// TIA Portal V15.1 export
// export: Created 2024-05-17T05:39:00.3704573Z, ExportSetting WithDefaults, DisplayName Totally Integrated Automation Portal, DisplayVersion V15.1 Update 5, DisplayName TIA Portal Openness, DisplayVersion V15.1 Update 5, DisplayName SINAMICS Startdrive Advanced, DisplayVersion V15.1, DisplayName G130, G150, S120, S150, SINAMICS MV, S210, DisplayVersion V15.1, DisplayName G110M, G120, G120C, G120D, G120P, DisplayVersion V15.1, DisplayName STEP 7 Professional, DisplayVersion V15.1 Update 5, DisplayName STEP 7 Safety, DisplayVersion V15.1, DisplayName WinCC Professional, DisplayVersion V15.1 Update 5, DisplayName SIMATIC Visualization Architect, DisplayVersion V15.1
FUNCTION "209000NCP01AE" : Void   // FC253, FBD
TITLE = 209000NCP01AE
{ S7_Optimized_Access := 'FALSE' }
AUTHOR : VCC
NAME : LocFnc
VERSION : 0.1
// stored: AutoNumber false, IsIECCheckEnabled false, SetENOAutomatically False, UDAEnableTagReadback false
   VAR_OUTPUT
      O_AlarmA : Bool;   // Alarm A
      O_AlarmB : Bool;   // Alarm B
      O_AlarmC : Bool;   // Alarm C
      O_AlarmD : Bool;   // Alarm D
      O_AlarmABCondition : Bool;   // Alarms resetable
      H_IAnim : Word;   // For animation of icon
   END_VAR
BEGIN

REGION Network 1: **** --------------------- AE01 --------------------- ****
END_REGION

REGION Network 2: **** 2.2 Alarms - Alarm generation **** AE01E1QM1 - AE01 EG1 - Overload protection power supply 24VDC
   // AE01 EG1 - Overload protection power supply 24VDC
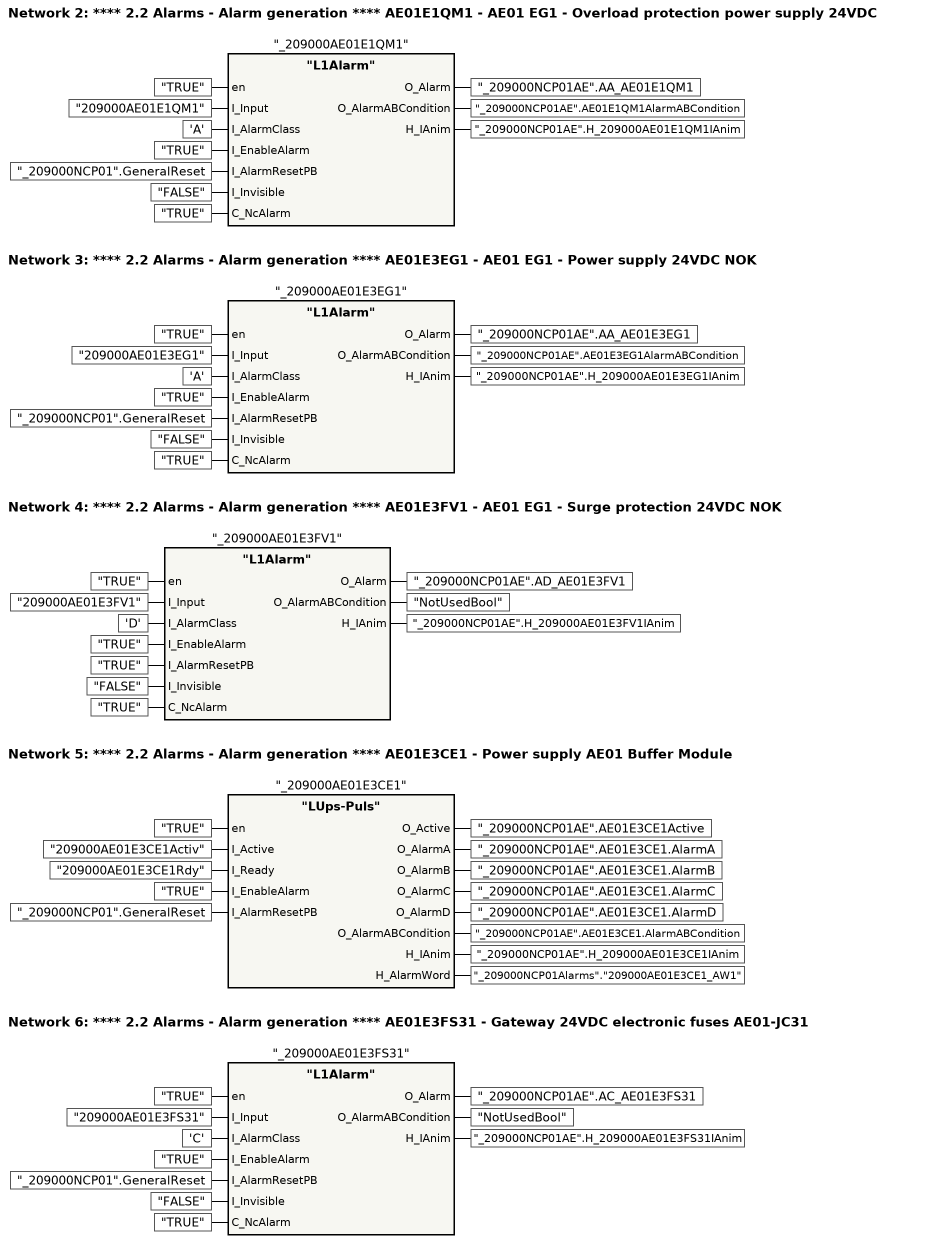
   IF "TRUE" THEN
       "_209000AE01E1QM1"(I_Input := "209000AE01E1QM1",   // "L1Alarm"
                          I_AlarmClass := 'A',
                          I_EnableAlarm := "TRUE",
                          I_AlarmResetPB := "_209000NCP01".GeneralReset,
                          I_Invisible := "FALSE",
                          C_NcAlarm := "TRUE",
                          O_Alarm => "_209000NCP01AE".AA_AE01E1QM1,
                          O_AlarmABCondition => "_209000NCP01AE".AE01E1QM1AlarmABCondition,
                          H_IAnim => "_209000NCP01AE".H_209000AE01E1QM1IAnim);
   END_IF;
END_REGION

REGION Network 3: **** 2.2 Alarms - Alarm generation **** AE01E3EG1 - AE01 EG1 - Power supply 24VDC NOK
   // AE01 EG1 - Power supply 24VDC NOK
   IF "TRUE" THEN
       "_209000AE01E3EG1"(I_Input := "209000AE01E3EG1",   // "L1Alarm"
                          I_AlarmClass := 'A',
                          I_EnableAlarm := "TRUE",
                          I_AlarmResetPB := "_209000NCP01".GeneralReset,
                          I_Invisible := "FALSE",
                          C_NcAlarm := "TRUE",
                          O_Alarm => "_209000NCP01AE".AA_AE01E3EG1,
                          O_AlarmABCondition => "_209000NCP01AE".AE01E3EG1AlarmABCondition,
                          H_IAnim => "_209000NCP01AE".H_209000AE01E3EG1IAnim);
   END_IF;
END_REGION

REGION Network 4: **** 2.2 Alarms - Alarm generation **** AE01E3FV1 - AE01 EG1 - Surge protection 24VDC NOK
   // AE01 EG1 - Surge protection 24VDC NOK
   IF "TRUE" THEN
       "_209000AE01E3FV1"(I_Input := "209000AE01E3FV1",   // "L1Alarm"
                          I_AlarmClass := 'D',
                          I_EnableAlarm := "TRUE",
                          I_AlarmResetPB := "TRUE",
                          I_Invisible := "FALSE",
                          C_NcAlarm := "TRUE",
                          O_Alarm => "_209000NCP01AE".AD_AE01E3FV1,
                          O_AlarmABCondition => "NotUsedBool",
                          H_IAnim => "_209000NCP01AE".H_209000AE01E3FV1IAnim);
   END_IF;
END_REGION

REGION Network 5: **** 2.2 Alarms - Alarm generation **** AE01E3CE1 - Power supply AE01 Buffer Module
   // Power supply  AE01 Buffer Module
   IF "TRUE" THEN
       "_209000AE01E3CE1"(I_Active := "209000AE01E3CE1Activ",   // "LUps-Puls"
                          I_Ready := "209000AE01E3CE1Rdy",
                          I_EnableAlarm := "TRUE",
                          I_AlarmResetPB := "_209000NCP01".GeneralReset,
                          O_Active => "_209000NCP01AE".AE01E3CE1Active,
                          O_AlarmA => "_209000NCP01AE".AE01E3CE1.AlarmA,
                          O_AlarmB => "_209000NCP01AE".AE01E3CE1.AlarmB,
                          O_AlarmC => "_209000NCP01AE".AE01E3CE1.AlarmC,
                          O_AlarmD => "_209000NCP01AE".AE01E3CE1.AlarmD,
                          O_AlarmABCondition => "_209000NCP01AE".AE01E3CE1.AlarmABCondition,
                          H_IAnim => "_209000NCP01AE".H_209000AE01E3CE1IAnim,
                          H_AlarmWord => "_209000NCP01Alarms"."209000AE01E3CE1_AW1");
   END_IF;
END_REGION

REGION Network 6: **** 2.2 Alarms - Alarm generation **** AE01E3FS31 - Gateway 24VDC electronic fuses AE01-JC31
   // Gateway 24VDC electronic fuses AE01-JC31
   IF "TRUE" THEN
       "_209000AE01E3FS31"(I_Input := "209000AE01E3FS31",   // "L1Alarm"
                           I_AlarmClass := 'C',
                           I_EnableAlarm := "TRUE",
                           I_AlarmResetPB := "_209000NCP01".GeneralReset,
                           I_Invisible := "FALSE",
                           C_NcAlarm := "TRUE",
                           O_Alarm => "_209000NCP01AE".AC_AE01E3FS31,
                           O_AlarmABCondition => "NotUsedBool",
                           H_IAnim => "_209000NCP01AE".H_209000AE01E3FS31IAnim);
   END_IF;
END_REGION

REGION Network 7: **** 2.2 Alarms - Alarm generation **** AE01E3FS01 // CH1 - 24VDC Fuse - General - PLC
   // 24VDC Fuse - General - PLC
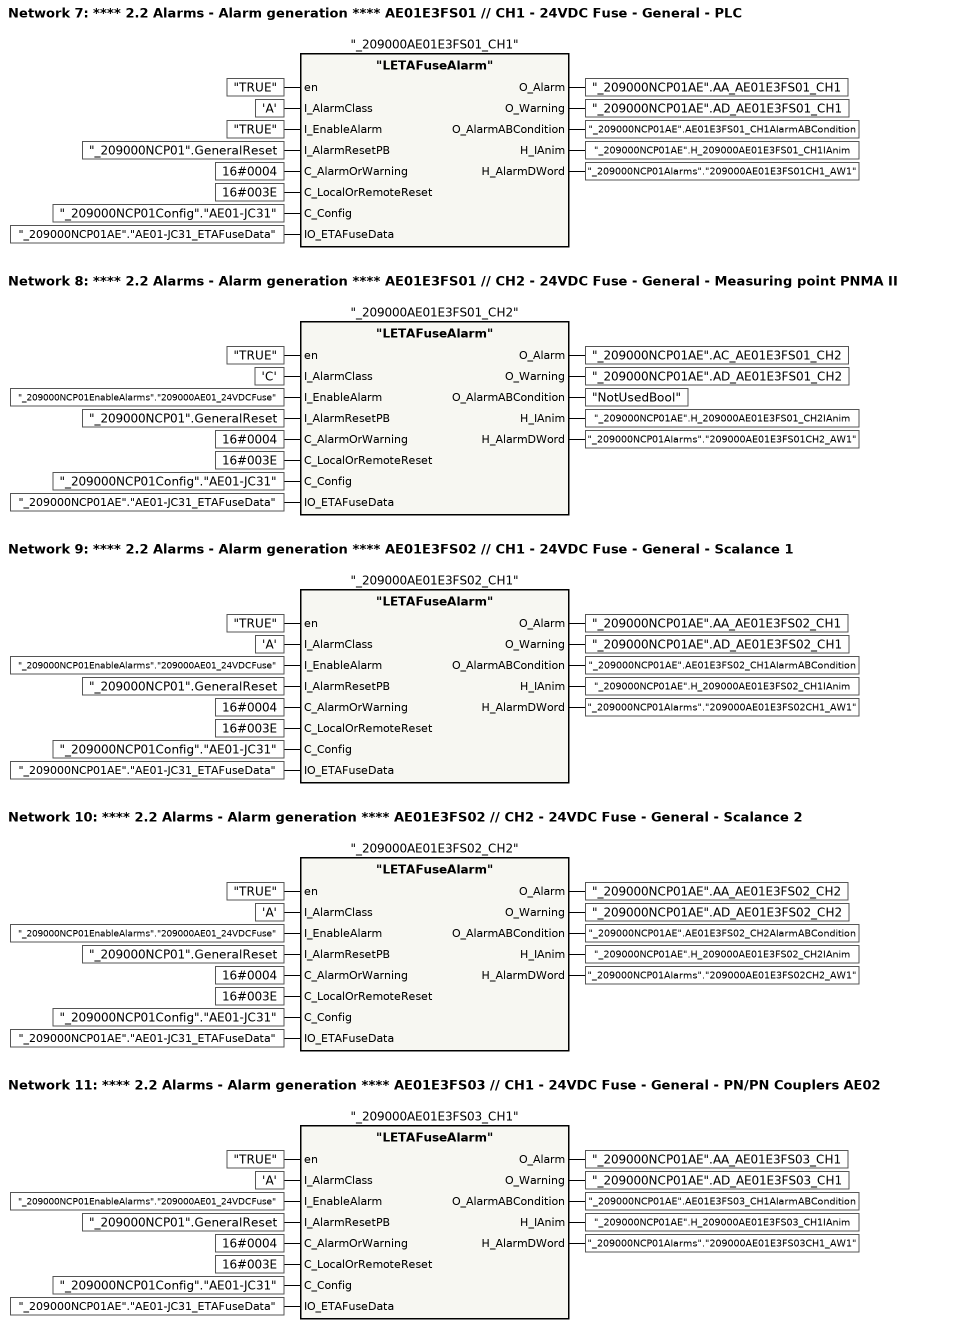
   IF "TRUE" THEN
       "_209000AE01E3FS01_CH1"(I_AlarmClass := 'A',   // "LETAFuseAlarm"
                               I_EnableAlarm := "TRUE",
                               I_AlarmResetPB := "_209000NCP01".GeneralReset,
                               C_AlarmOrWarning := 16#0004,
                               C_LocalOrRemoteReset := 16#003E,
                               C_Config := "_209000NCP01Config"."AE01-JC31",
                               IO_ETAFuseData := "_209000NCP01AE"."AE01-JC31_ETAFuseData",
                               O_Alarm => "_209000NCP01AE".AA_AE01E3FS01_CH1,
                               O_Warning => "_209000NCP01AE".AD_AE01E3FS01_CH1,
                               O_AlarmABCondition => "_209000NCP01AE".AE01E3FS01_CH1AlarmABCondition,
                               H_IAnim => "_209000NCP01AE".H_209000AE01E3FS01_CH1IAnim,
                               H_AlarmDWord => "_209000NCP01Alarms"."209000AE01E3FS01CH1_AW1");
   END_IF;
END_REGION

REGION Network 8: **** 2.2 Alarms - Alarm generation **** AE01E3FS01 // CH2 - 24VDC Fuse - General - Measuring point PNMA II
   // 24VDC Fuse - General - Measuring point PNMA II
   IF "TRUE" THEN
       "_209000AE01E3FS01_CH2"(I_AlarmClass := 'C',   // "LETAFuseAlarm"
                               I_EnableAlarm := "_209000NCP01EnableAlarms"."209000AE01_24VDCFuse",
                               I_AlarmResetPB := "_209000NCP01".GeneralReset,
                               C_AlarmOrWarning := 16#0004,
                               C_LocalOrRemoteReset := 16#003E,
                               C_Config := "_209000NCP01Config"."AE01-JC31",
                               IO_ETAFuseData := "_209000NCP01AE"."AE01-JC31_ETAFuseData",
                               O_Alarm => "_209000NCP01AE".AC_AE01E3FS01_CH2,
                               O_Warning => "_209000NCP01AE".AD_AE01E3FS01_CH2,
                               O_AlarmABCondition => "NotUsedBool",
                               H_IAnim => "_209000NCP01AE".H_209000AE01E3FS01_CH2IAnim,
                               H_AlarmDWord => "_209000NCP01Alarms"."209000AE01E3FS01CH2_AW1");
   END_IF;
END_REGION

REGION Network 9: **** 2.2 Alarms - Alarm generation **** AE01E3FS02 // CH1 - 24VDC Fuse - General - Scalance 1
   // 24VDC Fuse - General - Scalance 1
   IF "TRUE" THEN
       "_209000AE01E3FS02_CH1"(I_AlarmClass := 'A',   // "LETAFuseAlarm"
                               I_EnableAlarm := "_209000NCP01EnableAlarms"."209000AE01_24VDCFuse",
                               I_AlarmResetPB := "_209000NCP01".GeneralReset,
                               C_AlarmOrWarning := 16#0004,
                               C_LocalOrRemoteReset := 16#003E,
                               C_Config := "_209000NCP01Config"."AE01-JC31",
                               IO_ETAFuseData := "_209000NCP01AE"."AE01-JC31_ETAFuseData",
                               O_Alarm => "_209000NCP01AE".AA_AE01E3FS02_CH1,
                               O_Warning => "_209000NCP01AE".AD_AE01E3FS02_CH1,
                               O_AlarmABCondition => "_209000NCP01AE".AE01E3FS02_CH1AlarmABCondition,
                               H_IAnim => "_209000NCP01AE".H_209000AE01E3FS02_CH1IAnim,
                               H_AlarmDWord => "_209000NCP01Alarms"."209000AE01E3FS02CH1_AW1");
   END_IF;
END_REGION

REGION Network 10: **** 2.2 Alarms - Alarm generation **** AE01E3FS02 // CH2 - 24VDC Fuse - General - Scalance 2
   // 24VDC Fuse - General - Scalance 2
   IF "TRUE" THEN
       "_209000AE01E3FS02_CH2"(I_AlarmClass := 'A',   // "LETAFuseAlarm"
                               I_EnableAlarm := "_209000NCP01EnableAlarms"."209000AE01_24VDCFuse",
                               I_AlarmResetPB := "_209000NCP01".GeneralReset,
                               C_AlarmOrWarning := 16#0004,
                               C_LocalOrRemoteReset := 16#003E,
                               C_Config := "_209000NCP01Config"."AE01-JC31",
                               IO_ETAFuseData := "_209000NCP01AE"."AE01-JC31_ETAFuseData",
                               O_Alarm => "_209000NCP01AE".AA_AE01E3FS02_CH2,
                               O_Warning => "_209000NCP01AE".AD_AE01E3FS02_CH2,
                               O_AlarmABCondition => "_209000NCP01AE".AE01E3FS02_CH2AlarmABCondition,
                               H_IAnim => "_209000NCP01AE".H_209000AE01E3FS02_CH2IAnim,
                               H_AlarmDWord => "_209000NCP01Alarms"."209000AE01E3FS02CH2_AW1");
   END_IF;
END_REGION

REGION Network 11: **** 2.2 Alarms - Alarm generation **** AE01E3FS03 // CH1 - 24VDC Fuse - General - PN/PN Couplers AE02
   // 24VDC Fuse - General - PN/PN Couplers AE02
   IF "TRUE" THEN
       "_209000AE01E3FS03_CH1"(I_AlarmClass := 'A',   // "LETAFuseAlarm"
                               I_EnableAlarm := "_209000NCP01EnableAlarms"."209000AE01_24VDCFuse",
                               I_AlarmResetPB := "_209000NCP01".GeneralReset,
                               C_AlarmOrWarning := 16#0004,
                               C_LocalOrRemoteReset := 16#003E,
                               C_Config := "_209000NCP01Config"."AE01-JC31",
                               IO_ETAFuseData := "_209000NCP01AE"."AE01-JC31_ETAFuseData",
                               O_Alarm => "_209000NCP01AE".AA_AE01E3FS03_CH1,
                               O_Warning => "_209000NCP01AE".AD_AE01E3FS03_CH1,
                               O_AlarmABCondition => "_209000NCP01AE".AE01E3FS03_CH1AlarmABCondition,
                               H_IAnim => "_209000NCP01AE".H_209000AE01E3FS03_CH1IAnim,
                               H_AlarmDWord => "_209000NCP01Alarms"."209000AE01E3FS03CH1_AW1");
   END_IF;
END_REGION

REGION Network 12: **** 2.2 Alarms - Alarm generation **** AE01E3FS03 // CH2 - 24VDC Fuse - General - Busnode + Com. PLC212
   // 24VDC Fuse - General - Busnode + Com. PLC212
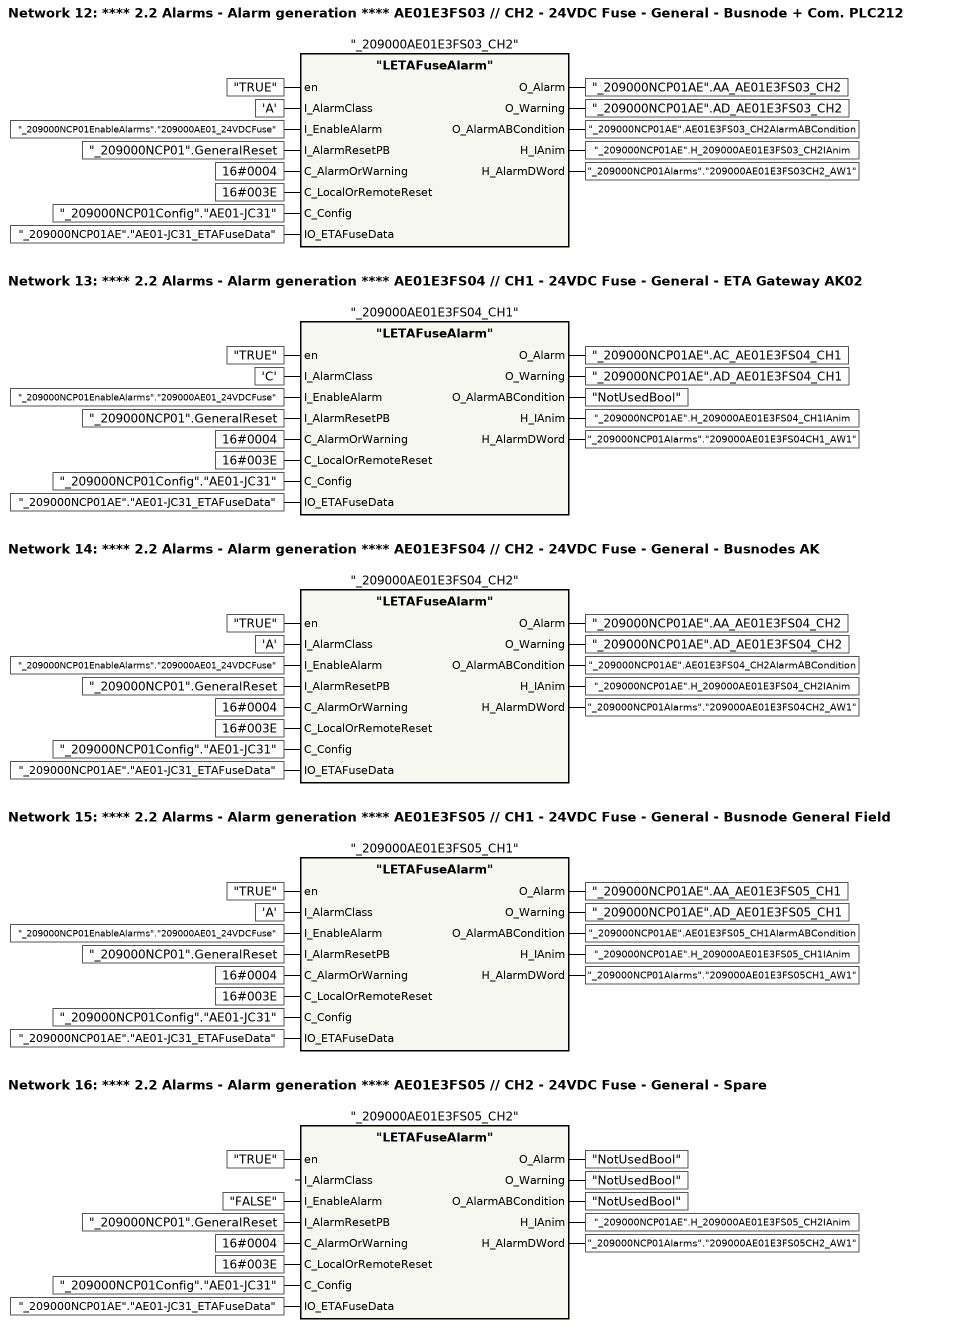
   IF "TRUE" THEN
       "_209000AE01E3FS03_CH2"(I_AlarmClass := 'A',   // "LETAFuseAlarm"
                               I_EnableAlarm := "_209000NCP01EnableAlarms"."209000AE01_24VDCFuse",
                               I_AlarmResetPB := "_209000NCP01".GeneralReset,
                               C_AlarmOrWarning := 16#0004,
                               C_LocalOrRemoteReset := 16#003E,
                               C_Config := "_209000NCP01Config"."AE01-JC31",
                               IO_ETAFuseData := "_209000NCP01AE"."AE01-JC31_ETAFuseData",
                               O_Alarm => "_209000NCP01AE".AA_AE01E3FS03_CH2,
                               O_Warning => "_209000NCP01AE".AD_AE01E3FS03_CH2,
                               O_AlarmABCondition => "_209000NCP01AE".AE01E3FS03_CH2AlarmABCondition,
                               H_IAnim => "_209000NCP01AE".H_209000AE01E3FS03_CH2IAnim,
                               H_AlarmDWord => "_209000NCP01Alarms"."209000AE01E3FS03CH2_AW1");
   END_IF;
END_REGION

REGION Network 13: **** 2.2 Alarms - Alarm generation **** AE01E3FS04 // CH1 - 24VDC Fuse - General - ETA Gateway AK02
   // 24VDC Fuse - General - ETA Gateway AK02
   IF "TRUE" THEN
       "_209000AE01E3FS04_CH1"(I_AlarmClass := 'C',   // "LETAFuseAlarm"
                               I_EnableAlarm := "_209000NCP01EnableAlarms"."209000AE01_24VDCFuse",
                               I_AlarmResetPB := "_209000NCP01".GeneralReset,
                               C_AlarmOrWarning := 16#0004,
                               C_LocalOrRemoteReset := 16#003E,
                               C_Config := "_209000NCP01Config"."AE01-JC31",
                               IO_ETAFuseData := "_209000NCP01AE"."AE01-JC31_ETAFuseData",
                               O_Alarm => "_209000NCP01AE".AC_AE01E3FS04_CH1,
                               O_Warning => "_209000NCP01AE".AD_AE01E3FS04_CH1,
                               O_AlarmABCondition => "NotUsedBool",
                               H_IAnim => "_209000NCP01AE".H_209000AE01E3FS04_CH1IAnim,
                               H_AlarmDWord => "_209000NCP01Alarms"."209000AE01E3FS04CH1_AW1");
   END_IF;
END_REGION

REGION Network 14: **** 2.2 Alarms - Alarm generation **** AE01E3FS04 // CH2 - 24VDC Fuse - General - Busnodes AK
   // 24VDC Fuse - General - Busnodes AK
   IF "TRUE" THEN
       "_209000AE01E3FS04_CH2"(I_AlarmClass := 'A',   // "LETAFuseAlarm"
                               I_EnableAlarm := "_209000NCP01EnableAlarms"."209000AE01_24VDCFuse",
                               I_AlarmResetPB := "_209000NCP01".GeneralReset,
                               C_AlarmOrWarning := 16#0004,
                               C_LocalOrRemoteReset := 16#003E,
                               C_Config := "_209000NCP01Config"."AE01-JC31",
                               IO_ETAFuseData := "_209000NCP01AE"."AE01-JC31_ETAFuseData",
                               O_Alarm => "_209000NCP01AE".AA_AE01E3FS04_CH2,
                               O_Warning => "_209000NCP01AE".AD_AE01E3FS04_CH2,
                               O_AlarmABCondition => "_209000NCP01AE".AE01E3FS04_CH2AlarmABCondition,
                               H_IAnim => "_209000NCP01AE".H_209000AE01E3FS04_CH2IAnim,
                               H_AlarmDWord => "_209000NCP01Alarms"."209000AE01E3FS04CH2_AW1");
   END_IF;
END_REGION

REGION Network 15: **** 2.2 Alarms - Alarm generation **** AE01E3FS05 // CH1 - 24VDC Fuse - General - Busnode General Field
   // 24VDC Fuse - General - Busnode General Field
   IF "TRUE" THEN
       "_209000AE01E3FS05_CH1"(I_AlarmClass := 'A',   // "LETAFuseAlarm"
                               I_EnableAlarm := "_209000NCP01EnableAlarms"."209000AE01_24VDCFuse",
                               I_AlarmResetPB := "_209000NCP01".GeneralReset,
                               C_AlarmOrWarning := 16#0004,
                               C_LocalOrRemoteReset := 16#003E,
                               C_Config := "_209000NCP01Config"."AE01-JC31",
                               IO_ETAFuseData := "_209000NCP01AE"."AE01-JC31_ETAFuseData",
                               O_Alarm => "_209000NCP01AE".AA_AE01E3FS05_CH1,
                               O_Warning => "_209000NCP01AE".AD_AE01E3FS05_CH1,
                               O_AlarmABCondition => "_209000NCP01AE".AE01E3FS05_CH1AlarmABCondition,
                               H_IAnim => "_209000NCP01AE".H_209000AE01E3FS05_CH1IAnim,
                               H_AlarmDWord => "_209000NCP01Alarms"."209000AE01E3FS05CH1_AW1");
   END_IF;
END_REGION

REGION Network 16: **** 2.2 Alarms - Alarm generation **** AE01E3FS05 // CH2 - 24VDC Fuse - General - Spare
   // 24VDC Fuse - General - Spare
   IF "TRUE" THEN
       "_209000AE01E3FS05_CH2"(I_EnableAlarm := "FALSE",   // "LETAFuseAlarm"
                               I_AlarmResetPB := "_209000NCP01".GeneralReset,
                               C_AlarmOrWarning := 16#0004,
                               C_LocalOrRemoteReset := 16#003E,
                               C_Config := "_209000NCP01Config"."AE01-JC31",
                               IO_ETAFuseData := "_209000NCP01AE"."AE01-JC31_ETAFuseData",
                               O_Alarm => "NotUsedBool",
                               O_Warning => "NotUsedBool",
                               O_AlarmABCondition => "NotUsedBool",
                               H_IAnim => "_209000NCP01AE".H_209000AE01E3FS05_CH2IAnim,
                               H_AlarmDWord => "_209000NCP01Alarms"."209000AE01E3FS05CH2_AW1");
   END_IF;
END_REGION

REGION Network 17: **** 2.2 Alarms - Alarm generation **** AE01EL1 - Fault heat exchanger cabinet AE01
   // Fault heat exchanger cabinet AE01
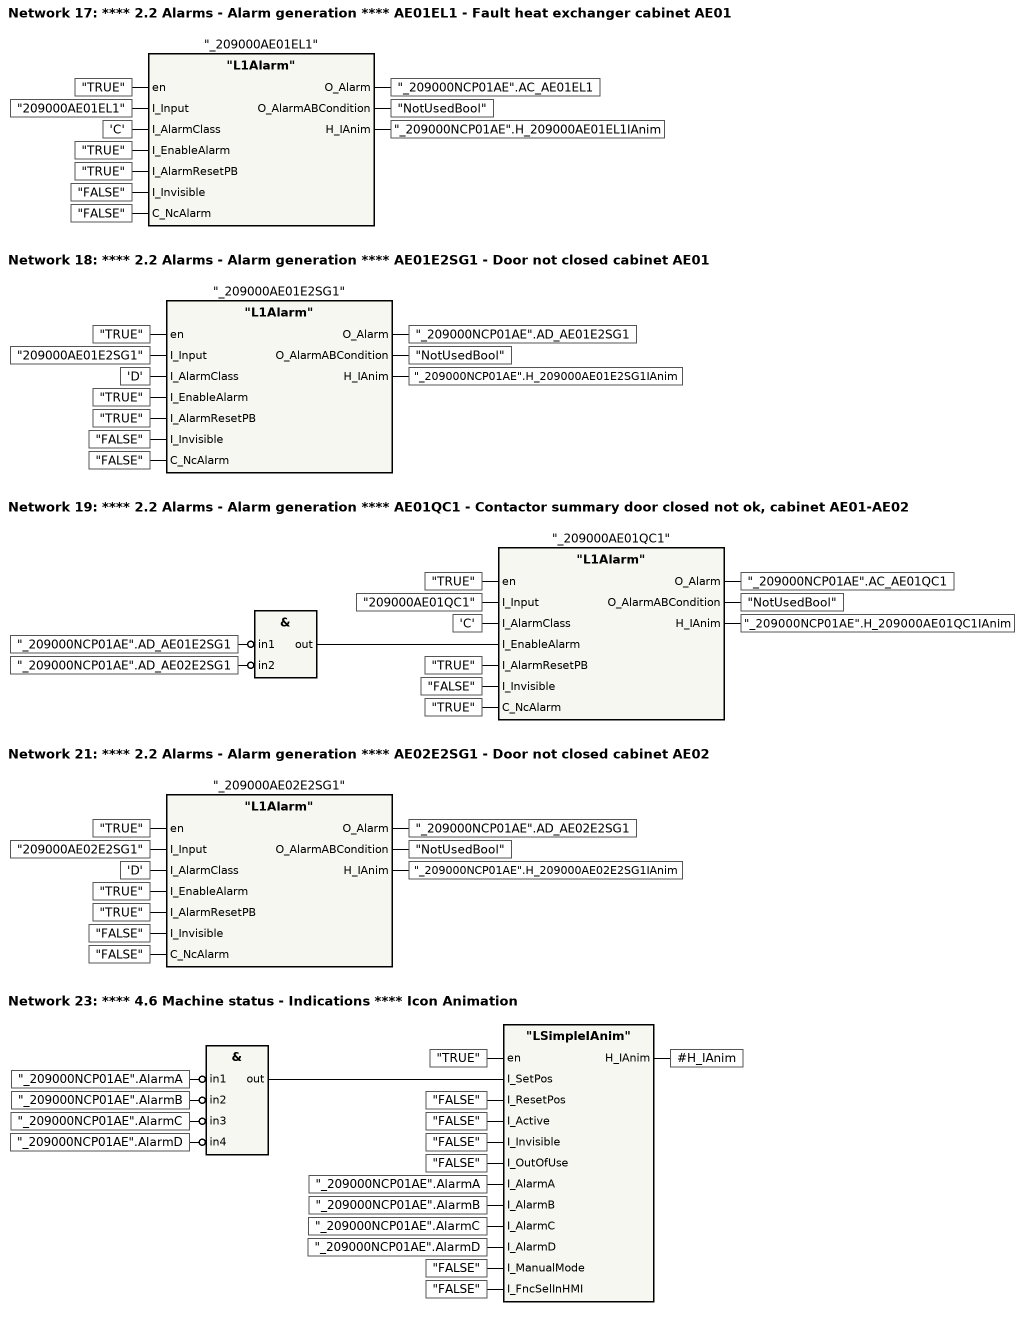
   IF "TRUE" THEN
       "_209000AE01EL1"(I_Input := "209000AE01EL1",   // "L1Alarm"
                        I_AlarmClass := 'C',
                        I_EnableAlarm := "TRUE",
                        I_AlarmResetPB := "TRUE",
                        I_Invisible := "FALSE",
                        C_NcAlarm := "FALSE",
                        O_Alarm => "_209000NCP01AE".AC_AE01EL1,
                        O_AlarmABCondition => "NotUsedBool",
                        H_IAnim => "_209000NCP01AE".H_209000AE01EL1IAnim);
   END_IF;
END_REGION

REGION Network 18: **** 2.2 Alarms - Alarm generation **** AE01E2SG1 - Door not closed cabinet AE01
   // Door not closed cabinet AE01
   IF "TRUE" THEN
       "_209000AE01E2SG1"(I_Input := "209000AE01E2SG1",   // "L1Alarm"
                          I_AlarmClass := 'D',
                          I_EnableAlarm := "TRUE",
                          I_AlarmResetPB := "TRUE",
                          I_Invisible := "FALSE",
                          C_NcAlarm := "FALSE",
                          O_Alarm => "_209000NCP01AE".AD_AE01E2SG1,
                          O_AlarmABCondition => "NotUsedBool",
                          H_IAnim => "_209000NCP01AE".H_209000AE01E2SG1IAnim);
   END_IF;
END_REGION

REGION Network 19: **** 2.2 Alarms - Alarm generation **** AE01QC1 - Contactor summary door closed not ok, cabinet AE01-AE02
   // Contactor summary door closed not ok, cabinet AE01-AE02
   IF "TRUE" THEN
       "_209000AE01QC1"(I_Input := "209000AE01QC1",   // "L1Alarm"
                        I_AlarmClass := 'C',
                        I_EnableAlarm := NOT "_209000NCP01AE".AD_AE01E2SG1 AND NOT "_209000NCP01AE".AD_AE02E2SG1,
                        I_AlarmResetPB := "TRUE",
                        I_Invisible := "FALSE",
                        C_NcAlarm := "TRUE",
                        O_Alarm => "_209000NCP01AE".AC_AE01QC1,
                        O_AlarmABCondition => "NotUsedBool",
                        H_IAnim => "_209000NCP01AE".H_209000AE01QC1IAnim);
   END_IF;
END_REGION

REGION Network 20: **** --------------------- AE02 --------------------- ****
END_REGION

REGION Network 21: **** 2.2 Alarms - Alarm generation **** AE02E2SG1 - Door not closed cabinet AE02
   // Door not closed cabinet AE02
   IF "TRUE" THEN
       "_209000AE02E2SG1"(I_Input := "209000AE02E2SG1",   // "L1Alarm"
                          I_AlarmClass := 'D',
                          I_EnableAlarm := "TRUE",
                          I_AlarmResetPB := "TRUE",
                          I_Invisible := "FALSE",
                          C_NcAlarm := "FALSE",
                          O_Alarm => "_209000NCP01AE".AD_AE02E2SG1,
                          O_AlarmABCondition => "NotUsedBool",
                          H_IAnim => "_209000NCP01AE".H_209000AE02E2SG1IAnim);
   END_IF;
END_REGION

REGION Network 22: **** -------------------------------------------------- ****
END_REGION

REGION Network 23: **** 4.6 Machine status - Indications **** Icon Animation
   // Animation for icon
   IF "TRUE" THEN
       "LSimpleIAnim"(I_SetPos := NOT "_209000NCP01AE".AlarmA AND NOT "_209000NCP01AE".AlarmB AND NOT "_209000NCP01AE".AlarmC AND NOT "_209000NCP01AE".AlarmD,
                      I_ResetPos := "FALSE",
                      I_Active := "FALSE",
                      I_Invisible := "FALSE",
                      I_OutOfUse := "FALSE",
                      I_AlarmA := "_209000NCP01AE".AlarmA,
                      I_AlarmB := "_209000NCP01AE".AlarmB,
                      I_AlarmC := "_209000NCP01AE".AlarmC,
                      I_AlarmD := "_209000NCP01AE".AlarmD,
                      I_ManualMode := "FALSE",
                      I_FncSelInHMI := "FALSE",
                      H_IAnim => #H_IAnim);
   END_IF;
END_REGION

REGION Network 24: **** 4.6 - Machine status - Indications **** Animation
   // Animation
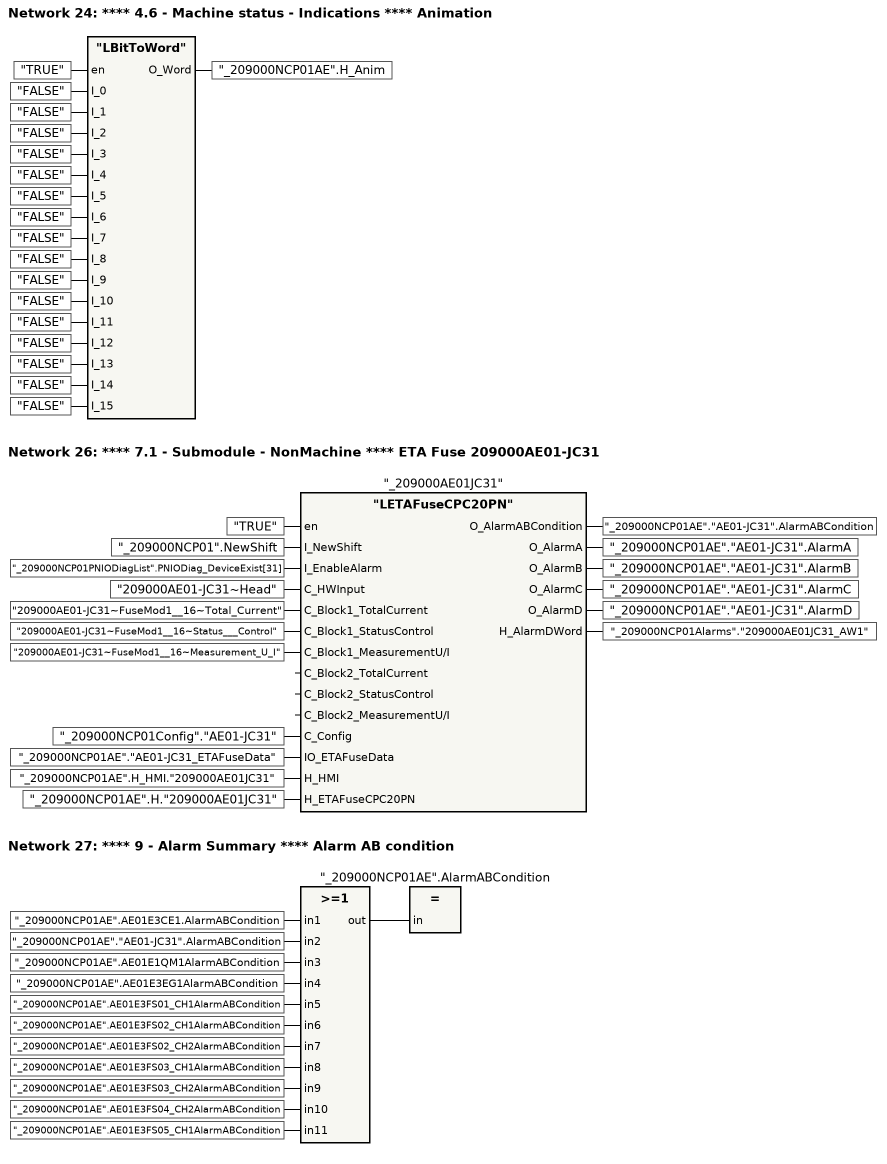
   IF "TRUE" THEN
       "LBitToWord"(I_0 := "FALSE",
                    I_1 := "FALSE",
                    I_2 := "FALSE",
                    I_3 := "FALSE",
                    I_4 := "FALSE",
                    I_5 := "FALSE",
                    I_6 := "FALSE",
                    I_7 := "FALSE",
                    I_8 := "FALSE",
                    I_9 := "FALSE",
                    I_10 := "FALSE",
                    I_11 := "FALSE",
                    I_12 := "FALSE",
                    I_13 := "FALSE",
                    I_14 := "FALSE",
                    I_15 := "FALSE",
                    O_Word => "_209000NCP01AE".H_Anim);
   END_IF;
END_REGION

NETWORK
TITLE = **** 4.6 - Machine Status - Indications **** Animation DB number
// DB number
      OPN   "_209000NCP01AE";
      L     DBNO;
      T     "_209000NCP01AE".H_DBnr;

REGION Network 26: **** 7.1 - Submodule - NonMachine **** ETA Fuse 209000AE01-JC31
   IF "TRUE" THEN
       "_209000AE01JC31"(I_NewShift := "_209000NCP01".NewShift,   // "LETAFuseCPC20PN"
                         I_EnableAlarm := "_209000NCP01PNIODiagList".PNIODiag_DeviceExist[31],
                         C_HWInput := "209000AE01-JC31~Head",
                         C_Block1_TotalCurrent := "209000AE01-JC31~FuseMod1__16~Total_Current",
                         C_Block1_StatusControl := "209000AE01-JC31~FuseMod1__16~Status___Control",
                         "C_Block1_MeasurementU/I" := "209000AE01-JC31~FuseMod1__16~Measurement_U_I",
                         C_Config := "_209000NCP01Config"."AE01-JC31",
                         IO_ETAFuseData := "_209000NCP01AE"."AE01-JC31_ETAFuseData",
                         H_HMI := "_209000NCP01AE".H_HMI."209000AE01JC31",
                         H_ETAFuseCPC20PN := "_209000NCP01AE".H."209000AE01JC31",
                         O_AlarmABCondition => "_209000NCP01AE"."AE01-JC31".AlarmABCondition,
                         O_AlarmA => "_209000NCP01AE"."AE01-JC31".AlarmA,
                         O_AlarmB => "_209000NCP01AE"."AE01-JC31".AlarmB,
                         O_AlarmC => "_209000NCP01AE"."AE01-JC31".AlarmC,
                         O_AlarmD => "_209000NCP01AE"."AE01-JC31".AlarmD,
                         H_AlarmDWord => "_209000NCP01Alarms"."209000AE01JC31_AW1");
   END_IF;
END_REGION

REGION Network 27: **** 9 - Alarm Summary **** Alarm AB condition
   // Alarm AB condition
   "_209000NCP01AE".AlarmABCondition := "_209000NCP01AE".AE01E3CE1.AlarmABCondition OR "_209000NCP01AE"."AE01-JC31".AlarmABCondition OR "_209000NCP01AE".AE01E1QM1AlarmABCondition OR "_209000NCP01AE".AE01E3EG1AlarmABCondition OR "_209000NCP01AE".AE01E3FS01_CH1AlarmABCondition OR "_209000NCP01AE".AE01E3FS02_CH1AlarmABCondition OR "_209000NCP01AE".AE01E3FS02_CH2AlarmABCondition OR "_209000NCP01AE".AE01E3FS03_CH1AlarmABCondition OR "_209000NCP01AE".AE01E3FS03_CH2AlarmABCondition OR "_209000NCP01AE".AE01E3FS04_CH2AlarmABCondition OR "_209000NCP01AE".AE01E3FS05_CH1AlarmABCondition;
END_REGION

REGION Network 28: **** 9 - Alarm Summary **** Alarm A
   // Summary of alarms A
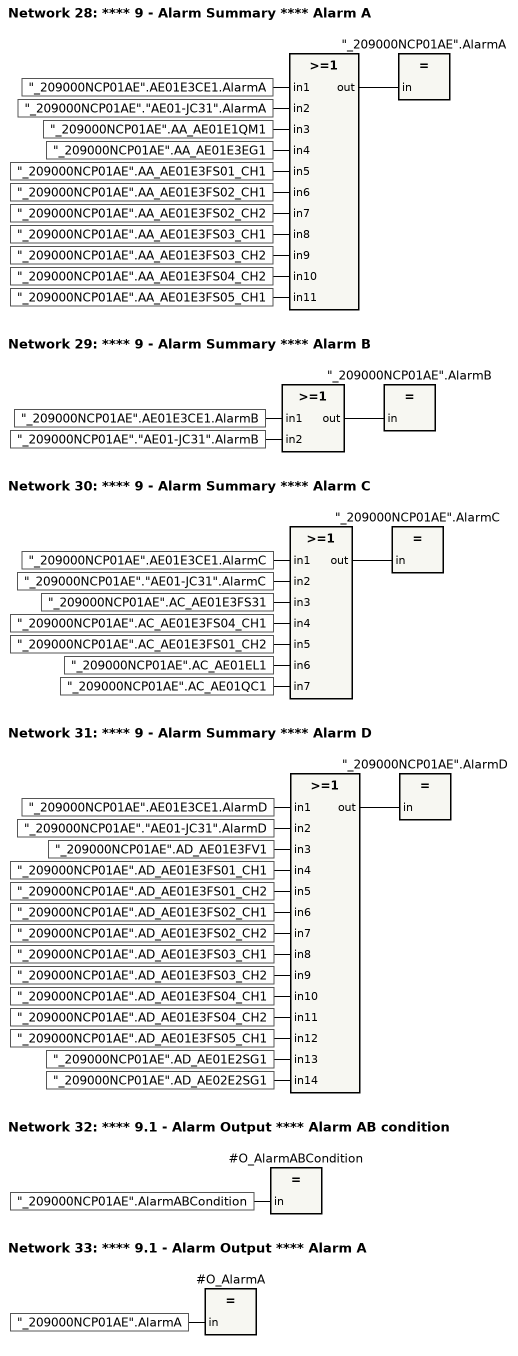
   "_209000NCP01AE".AlarmA := "_209000NCP01AE".AE01E3CE1.AlarmA OR "_209000NCP01AE"."AE01-JC31".AlarmA OR "_209000NCP01AE".AA_AE01E1QM1 OR "_209000NCP01AE".AA_AE01E3EG1 OR "_209000NCP01AE".AA_AE01E3FS01_CH1 OR "_209000NCP01AE".AA_AE01E3FS02_CH1 OR "_209000NCP01AE".AA_AE01E3FS02_CH2 OR "_209000NCP01AE".AA_AE01E3FS03_CH1 OR "_209000NCP01AE".AA_AE01E3FS03_CH2 OR "_209000NCP01AE".AA_AE01E3FS04_CH2 OR "_209000NCP01AE".AA_AE01E3FS05_CH1;
END_REGION

REGION Network 29: **** 9 - Alarm Summary **** Alarm B
   // Summary of alarms B
   "_209000NCP01AE".AlarmB := "_209000NCP01AE".AE01E3CE1.AlarmB OR "_209000NCP01AE"."AE01-JC31".AlarmB;
END_REGION

REGION Network 30: **** 9 - Alarm Summary **** Alarm C
   // Summary of alarms C
   "_209000NCP01AE".AlarmC := "_209000NCP01AE".AE01E3CE1.AlarmC OR "_209000NCP01AE"."AE01-JC31".AlarmC OR "_209000NCP01AE".AC_AE01E3FS31 OR "_209000NCP01AE".AC_AE01E3FS04_CH1 OR "_209000NCP01AE".AC_AE01E3FS01_CH2 OR "_209000NCP01AE".AC_AE01EL1 OR "_209000NCP01AE".AC_AE01QC1;
END_REGION

REGION Network 31: **** 9 - Alarm Summary **** Alarm D
   // Summary of alarms D
   "_209000NCP01AE".AlarmD := "_209000NCP01AE".AE01E3CE1.AlarmD OR "_209000NCP01AE"."AE01-JC31".AlarmD OR "_209000NCP01AE".AD_AE01E3FV1 OR "_209000NCP01AE".AD_AE01E3FS01_CH1 OR "_209000NCP01AE".AD_AE01E3FS01_CH2 OR "_209000NCP01AE".AD_AE01E3FS02_CH1 OR "_209000NCP01AE".AD_AE01E3FS02_CH2 OR "_209000NCP01AE".AD_AE01E3FS03_CH1 OR "_209000NCP01AE".AD_AE01E3FS03_CH2 OR "_209000NCP01AE".AD_AE01E3FS04_CH1 OR "_209000NCP01AE".AD_AE01E3FS04_CH2 OR "_209000NCP01AE".AD_AE01E3FS05_CH1 OR "_209000NCP01AE".AD_AE01E2SG1 OR "_209000NCP01AE".AD_AE02E2SG1;
END_REGION

REGION Network 32: **** 9.1 - Alarm Output **** Alarm AB condition
   // Alarm AB condition
   #O_AlarmABCondition := "_209000NCP01AE".AlarmABCondition;
END_REGION

REGION Network 33: **** 9.1 - Alarm Output **** Alarm A
   // Summary of alarms A
   #O_AlarmA := "_209000NCP01AE".AlarmA;
END_REGION

REGION Network 34: **** 9.1 - Alarm Output **** Alarm B
   // Summary of alarms B
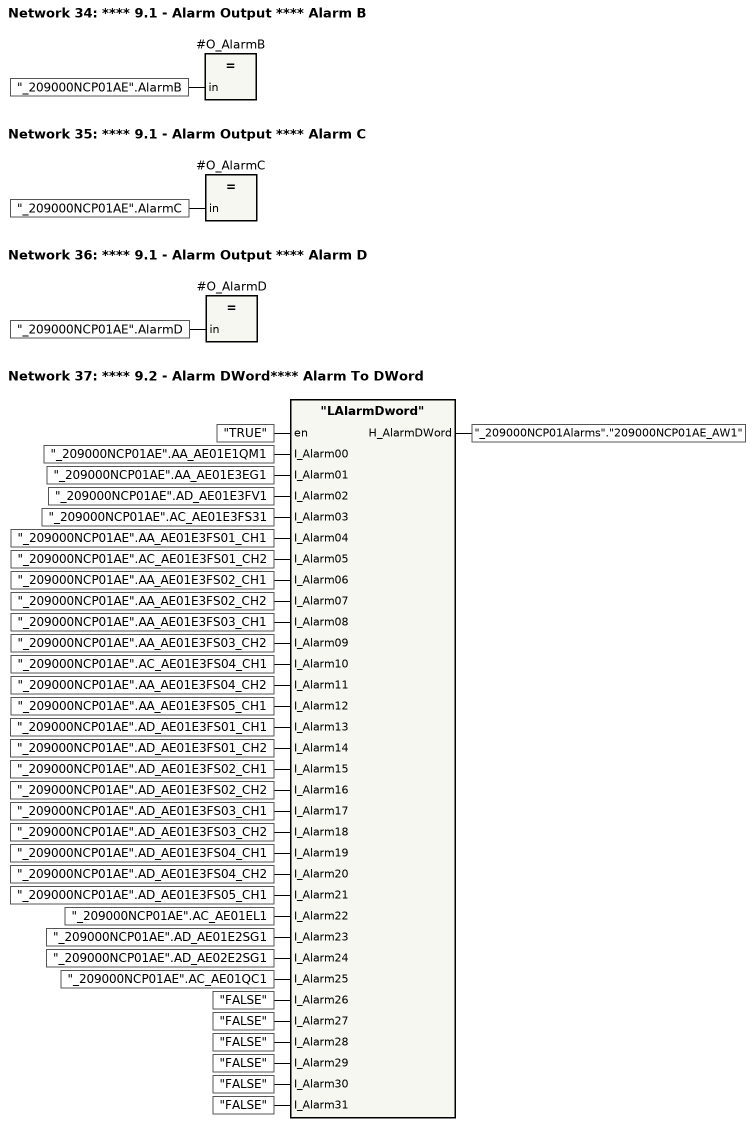
   #O_AlarmB := "_209000NCP01AE".AlarmB;
END_REGION

REGION Network 35: **** 9.1 - Alarm Output **** Alarm C
   // Summary of alarms C
   #O_AlarmC := "_209000NCP01AE".AlarmC;
END_REGION

REGION Network 36: **** 9.1 - Alarm Output **** Alarm D
   // Summary of alarms D
   #O_AlarmD := "_209000NCP01AE".AlarmD;
END_REGION

REGION Network 37: **** 9.2 - Alarm DWord**** Alarm To DWord
   // Alarm Word
   IF "TRUE" THEN
       "LAlarmDword"(I_Alarm00 := "_209000NCP01AE".AA_AE01E1QM1,
                     I_Alarm01 := "_209000NCP01AE".AA_AE01E3EG1,
                     I_Alarm02 := "_209000NCP01AE".AD_AE01E3FV1,
                     I_Alarm03 := "_209000NCP01AE".AC_AE01E3FS31,
                     I_Alarm04 := "_209000NCP01AE".AA_AE01E3FS01_CH1,
                     I_Alarm05 := "_209000NCP01AE".AC_AE01E3FS01_CH2,
                     I_Alarm06 := "_209000NCP01AE".AA_AE01E3FS02_CH1,
                     I_Alarm07 := "_209000NCP01AE".AA_AE01E3FS02_CH2,
                     I_Alarm08 := "_209000NCP01AE".AA_AE01E3FS03_CH1,
                     I_Alarm09 := "_209000NCP01AE".AA_AE01E3FS03_CH2,
                     I_Alarm10 := "_209000NCP01AE".AC_AE01E3FS04_CH1,
                     I_Alarm11 := "_209000NCP01AE".AA_AE01E3FS04_CH2,
                     I_Alarm12 := "_209000NCP01AE".AA_AE01E3FS05_CH1,
                     I_Alarm13 := "_209000NCP01AE".AD_AE01E3FS01_CH1,
                     I_Alarm14 := "_209000NCP01AE".AD_AE01E3FS01_CH2,
                     I_Alarm15 := "_209000NCP01AE".AD_AE01E3FS02_CH1,
                     I_Alarm16 := "_209000NCP01AE".AD_AE01E3FS02_CH2,
                     I_Alarm17 := "_209000NCP01AE".AD_AE01E3FS03_CH1,
                     I_Alarm18 := "_209000NCP01AE".AD_AE01E3FS03_CH2,
                     I_Alarm19 := "_209000NCP01AE".AD_AE01E3FS04_CH1,
                     I_Alarm20 := "_209000NCP01AE".AD_AE01E3FS04_CH2,
                     I_Alarm21 := "_209000NCP01AE".AD_AE01E3FS05_CH1,
                     I_Alarm22 := "_209000NCP01AE".AC_AE01EL1,
                     I_Alarm23 := "_209000NCP01AE".AD_AE01E2SG1,
                     I_Alarm24 := "_209000NCP01AE".AD_AE02E2SG1,
                     I_Alarm25 := "_209000NCP01AE".AC_AE01QC1,
                     I_Alarm26 := "FALSE",
                     I_Alarm27 := "FALSE",
                     I_Alarm28 := "FALSE",
                     I_Alarm29 := "FALSE",
                     I_Alarm30 := "FALSE",
                     I_Alarm31 := "FALSE",
                     H_AlarmDWord => "_209000NCP01Alarms"."209000NCP01AE_AW1");
   END_IF;
END_REGION
END_FUNCTION
